PROGRAM AxisPowerOn
VAR

END_VAR


//左臂-左电机-PowerOn
axis_LeftArm_Left_Power(
	Axis:= axis_LeftArm_Left, 
	Enable:= bAxis_LeftArm_Left_Enable, 
	Enable_Positive:= TRUE, 
	Enable_Negative:= TRUE, 
	Override:= , 
	BufferMode:= , 
	Options:= , 
	Status=> axis_LeftArm_Left_Power_Output.Done, 
	Busy=> , 
	Error=> , 
	ErrorID=> );
	
	
//左臂-右电机-PowerOn
axis_LeftArm_Right_Power(
	Axis:= axis_LeftArm_Right, 
	Enable:= bAxis_LeftArm_Right_Enable, 
	Enable_Positive:= TRUE, 
	Enable_Negative:= TRUE, 
	Override:= , 
	BufferMode:= , 
	Options:= , 
	Status=> axis_LeftArm_Right_Power_Output.Done, 
	Busy=> , 
	Error=> , 
	ErrorID=> );
	
axis_LeftArm_Lift_Power(
	Axis:= axis_LeftArm_Lift, 
	Enable:= bAxis_LeftArm_Lift_Enable, 
	Enable_Positive:= TRUE, 
	Enable_Negative:= TRUE, 
	Override:= , 
	BufferMode:= , 
	Options:= , 
	Status=> , 
	Busy=> , 
	Error=> , 
	ErrorID=> );

axis_LeftArm_Wrist_Power(
	Axis:= axis_LeftArm_Wrist, 
	Enable:= bAxis_LeftArm_Wrist_Enable, 
	Enable_Positive:= TRUE, 
	Enable_Negative:= TRUE, 
	Override:= , 
	BufferMode:= , 
	Options:= , 
	Status=> , 
	Busy=> , 
	Error=> , 
	ErrorID=> );




//右臂-左电机-PowerOn
axis_RightArm_Left_Power(
	Axis:= axis_RightArm_Left, 
	Enable:= bAxis_RightArm_Left_Enable, 
	Enable_Positive:= TRUE, 
	Enable_Negative:= TRUE, 
	Override:= , 
	BufferMode:= , 
	Options:= , 
	Status=> axis_RightArm_Left_Power_Output.Done, 
	Busy=> , 
	Error=> , 
	ErrorID=> );
	
	
//右臂-右电机-PowerOn
axis_RightArm_Right_Power(
	Axis:= axis_RightArm_Right, 
	Enable:= bAxis_RightArm_Right_Enable, 
	Enable_Positive:= TRUE, 
	Enable_Negative:= TRUE, 
	Override:= , 
	BufferMode:= , 
	Options:= , 
	Status=> axis_RightArm_Right_Power_Output.Done, 
	Busy=> , 
	Error=> , 
	ErrorID=> );

//右臂-升电机-Poweron
axis_RightArm_Lift_Power(
	Axis:= axis_RightArm_Lift, 
	Enable:= bAxis_RightArm_Lift_Enable, 
	Enable_Positive:= TRUE, 
	Enable_Negative:= TRUE, 
	Override:= , 
	BufferMode:= , 
	Options:= , 
	Status=> , 
	Busy=> , 
	Error=> , 
	ErrorID=> );

//右臂-腕电机-Poweron
axis_RightArm_Wrist_Power(
	Axis:= axis_RightArm_Wrist, 
	Enable:= bAxis_RightArm_Wrist_Enable, 
	Enable_Positive:= TRUE, 
	Enable_Negative:= TRUE, 
	Override:= , 
	BufferMode:= , 
	Options:= , 
	Status=> , 
	Busy=> , 
	Error=> , 
	ErrorID=> );
	


	
//大龙门-左电机-上电
axis_BigGate_Left_Power(
	Axis:= axis_BigGate_Left, 
	Enable:= bAxis_BigGate_Left_Enable, 
	Enable_Positive:= TRUE, 
	Enable_Negative:= TRUE, 
	Override:= , 
	BufferMode:= , 
	Options:= , 
	Status=> axis_BigGate_Left_Power_Output.Done, 
	Busy=> , 
	Error=> , 
	ErrorID=> );
	
//大龙门-右电机-上电	
axis_BigGate_Right_Power(
	Axis:= axis_BigGate_Right, 
	Enable:= bAxis_BigGate_Right_Enable, 
	Enable_Positive:= TRUE, 
	Enable_Negative:= TRUE, 
	Override:= , 
	BufferMode:= , 
	Options:= , 
	Status=> axis_BigGate_Right_Power_Output.Done, 
	Busy=> , 
	Error=> , 
	ErrorID=> );

//小龙门-左电机-上电	
axis_SmallGate_Left_Power(
	Axis:= axis_SmallGate_Left, 
	Enable:= bAxis_SmallGate_Left_Enable, 
	Enable_Positive:= TRUE, 
	Enable_Negative:= TRUE, 
	Override:= , 
	BufferMode:= , 
	Options:= , 
	Status=> axis_SmallGate_Left_Power_Output.Done, 
	Busy=> , 
	Error=> , 
	ErrorID=> );
	
//小龙门-右电机-上电	
axis_SmallGate_Right_Power(
	Axis:= axis_SmallGate_Right, 
	Enable:= bAxis_SmallGate_Right_Enable, 
	Enable_Positive:= TRUE, 
	Enable_Negative:= TRUE, 
	Override:= , 
	BufferMode:= , 
	Options:= , 
	Status=> axis_SmallGate_Right_Power_Output.Done, 
	Busy=> , 
	Error=> , 
	ErrorID=> );

//后龙门-左电机-上电	
axis_BackGate_Left_Power(
	Axis:= axis_BackGate_Left, 
	Enable:= bAxis_BackGate_Left_Enable, 
	Enable_Positive:= TRUE, 
	Enable_Negative:= TRUE, 
	Override:= , 
	BufferMode:= , 
	Options:= , 
	Status=> axis_BackGate_Left_Power_Output.Done, 
	Busy=> , 
	Error=> , 
	ErrorID=> );

//后龙门-右电机-上电
axis_BackGate_Right_Power(
	Axis:= axis_BackGate_Right, 
	Enable:= bAxis_BackGate_Right_Enable, 
	Enable_Positive:= TRUE, 
	Enable_Negative:= TRUE, 
	Override:= , 
	BufferMode:= , 
	Options:= , 
	Status=> axis_BackGate_Right_Power_Output.Done, 
	Busy=> , 
	Error=> , 
	ErrorID=> );

END_PROGRAM

(* stored: Version 1.1.0.1, ProductVersion 3.1.4024.14
   POU AxisPowerOn: Id {d29dff74-ccf9-49c6-a3da-29ff957c32cd}, SpecialFunc None *)
